// TIA Portal V20 export
DATA_BLOCK "zFNet_Data"   // DB403
// stored: Access Published, MemoryReserve 100, Namespace CITI_Logic
   VAR
      FNet_Data : Array[0..9] of "CITI_Logic.FlexNet_Data";
   END_VAR
BEGIN
END_DATA_BLOCK
